FUNCTION_BLOCK TEST_SERVICE_LIST
  {SET_ATTRIBUTE(OpcUa, SERVICE)}
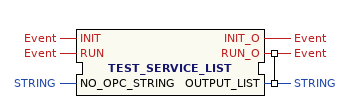
  EVENT_INPUT
    INIT;
    RUN;
  END_EVENT
  EVENT_OUTPUT
    INIT_O;
    RUN_O WITH OUTPUT_LIST;
  END_EVENT
  VAR_INPUT
    NO_OPC_STRING : STRING;
  END_VAR
  VAR_OUTPUT
    OUTPUT_LIST : STRING; {SET_ATTRIBUTE(OpcUa, Variable)}
  END_VAR
END_FUNCTION_BLOCK
